{attribute addProperty BoxType "KL2531"}
{attribute addProperty Id "StatusAT %I*USINT000PositionAT %I*UINT000ExtStatusAT %I*UINT000CtrlAT %Q*USINT000VelocityAT %Q*INT000ExtCtrlAT %Q*UINT000"}
{attribute addProperty CRC "2255117079"}
{attribute addProperty SizeInBites "0"}
{attribute addProperty SizeInBytes "0"}
TYPE Channel_866A5B17 :
STRUCT
	{attribute addProperty Name "Status"}
	Status AT %I* : USINT;
	{attribute addProperty Name "Position"}
	Position AT %I* : UINT;
	{attribute addProperty Name "ExtStatus"}
	ExtStatus AT %I* : UINT;
	{attribute addProperty Name "Ctrl"}
	Ctrl AT %Q* : USINT;
	{attribute addProperty Name "Velocity"}
	Velocity AT %Q* : INT;
	{attribute addProperty Name "ExtCtrl"}
	ExtCtrl AT %Q* : UINT;
END_STRUCT
END_TYPE

(* stored: Version 1.2.0.0, ProductVersion 3.1.4024.9
   DUT Channel_866A5B17: Id {bd328b1c-2e0a-48c4-bffb-e644feb3bf61} *)
